// TIA Portal V19 export
TYPE "LEXCHANGETRAY_typeSr1000ProfinetTelegram_readData128Byte"
// stored: Access Published
   STRUCT
      dataBytes : Array[0..127] of Byte;
      resultDataReadyCount : UInt;
      resultDataUpdateCount : UInt;
      resultDataSize : UInt;
      resultData0 : Char;
      resultData1 : Char;
      resultData2 : Char;
      resultData3 : Char;
      resultData4 : Char;
      resultData5 : Char;
      resultData6 : Char;
      resultData7 : Char;
      resultData8 : Char;
      resultData9 : Char;
      resultData10 : Char;
      resultData11 : Char;
      resultData12 : Char;
      resultData13 : Char;
      resultData14 : Char;
      resultData15 : Char;
   END_STRUCT;
END_TYPE
